// SIMATIC S7-200 project (STEP 7-Micro/WIN), CPU 224XP CN REL 02.01

SYMBOL_TABLE 用户定义1
键值输出1            I0.0
键值输出2            I0.1
键值输出3            I0.2
键值输出4            I0.3
传感器输出A           I0.4
传感器输出B           I0.5
传感器输出C           I0.6
传感器输出D           I0.7
手自动              I1.0
启停               I1.1
位置显示A            Q0.0
位置显示B            Q0.1
位置显示C            Q0.2
正传左行             Q0.3
反转右行             Q0.4
快速               Q0.5
慢速               Q0.6
报警               Q0.7
END_SYMBOL_TABLE

ORGANIZATION_BLOCK 主程序:OB1
TITLE=小车运动1A
// V0.0进入初始复位子程序控制位
// V0.1进入手动子程序控制位
// V0.2进入自动子程序控制位
// VW10初始复位控制用
// VW20手动控制用
// VW30自动控制用
BEGIN
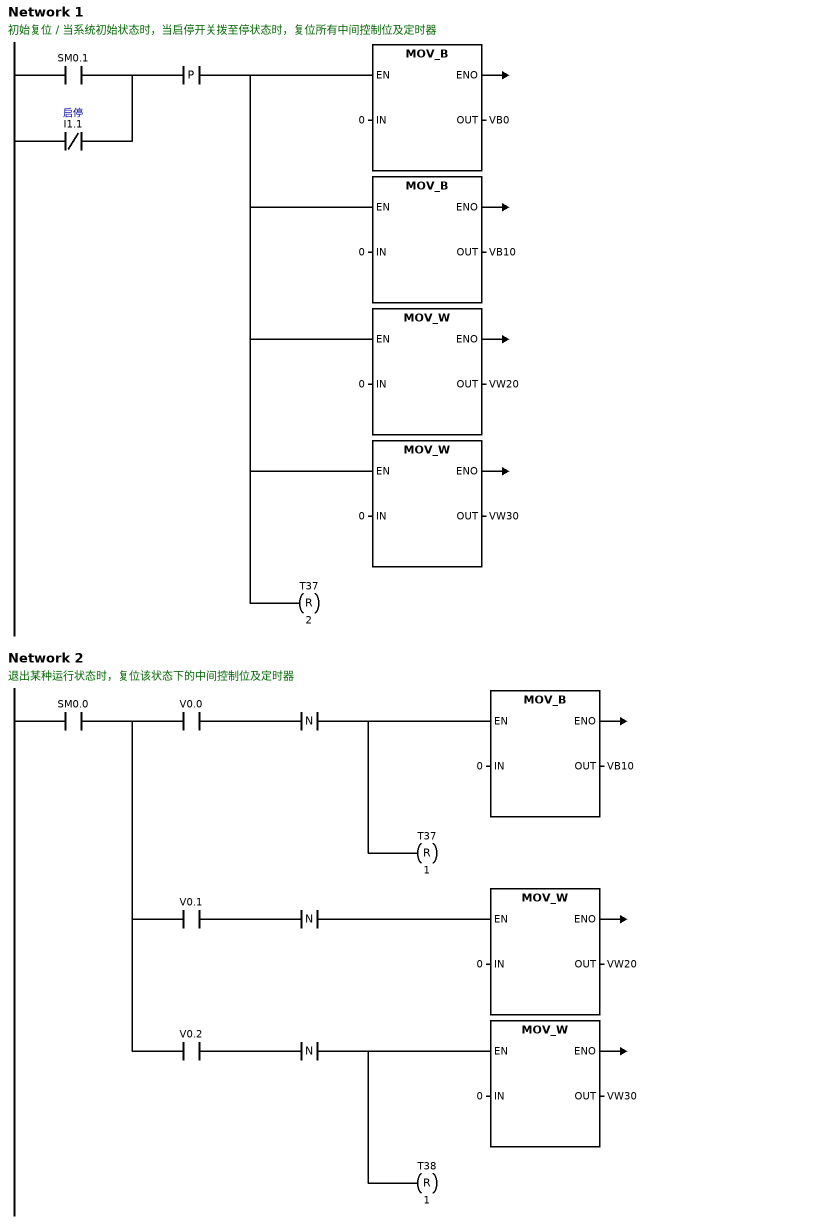
Network 1
// 初始复位
// 当系统初始状态时，当启停开关拨至停状态时，复位所有中间控制位及定时器
LD     SM0.1
ON     启停:I1.1
EU
MOVB   0, VB0
MOVB   0, VB10
MOVW   0, VW20
MOVW   0, VW30
R      T37, 2
Network 2
// 退出某种运行状态时，复位该状态下的中间控制位及定时器
LD     SM0.0
LPS
A      V0.0
ED
MOVB   0, VB10
R      T37, 1
LRD
A      V0.1
ED
MOVW   0, VW20
LPP
A      V0.2
ED
MOVW   0, VW30
R      T38, 1
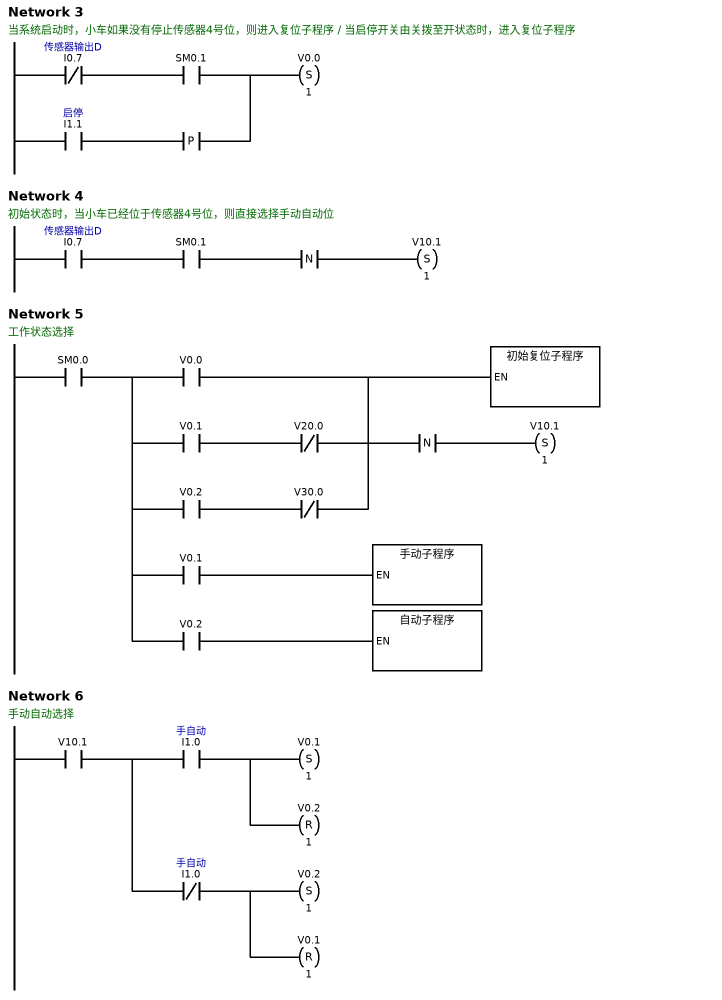
Network 3
// 当系统启动时，小车如果没有停止传感器4号位，则进入复位子程序
// 当启停开关由关拨至开状态时，进入复位子程序
LDN    传感器输出D:I0.7
A      SM0.1
LD     启停:I1.1
EU
OLD
S      V0.0, 1
Network 4
// 初始状态时，当小车已经位于传感器4号位，则直接选择手动自动位
LD     传感器输出D:I0.7
A      SM0.1
ED
S      V10.1, 1
Network 5
// 工作状态选择
LD     SM0.0
LPS
LD     V0.0
LD     V0.1
AN     V20.0
OLD
LD     V0.2
AN     V30.0
OLD
ALD
CALL   初始复位子程序:SBR0
ED
S      V10.1, 1
LPP
LPS
A      V0.1
CALL   手动子程序:SBR1
LPP
A      V0.2
CALL   自动子程序:SBR2
Network 6
// 手动自动选择
LD     V10.1
LPS
A      手自动:I1.0
S      V0.1, 1
R      V0.2, 1
LPP
AN     手自动:I1.0
S      V0.2, 1
R      V0.1, 1
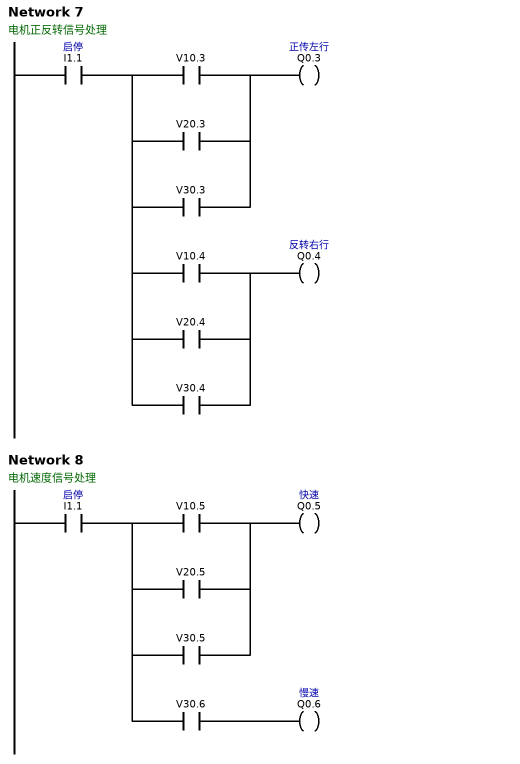
Network 7
// 电机正反转信号处理
LD     启停:I1.1
LPS
LD     V10.3
O      V20.3
O      V30.3
ALD
=      正传左行:Q0.3
LPP
LD     V10.4
O      V20.4
O      V30.4
ALD
=      反转右行:Q0.4
Network 8
// 电机速度信号处理
LD     启停:I1.1
LPS
LD     V10.5
O      V20.5
O      V30.5
ALD
=      快速:Q0.5
LPP
A      V30.6
=      慢速:Q0.6
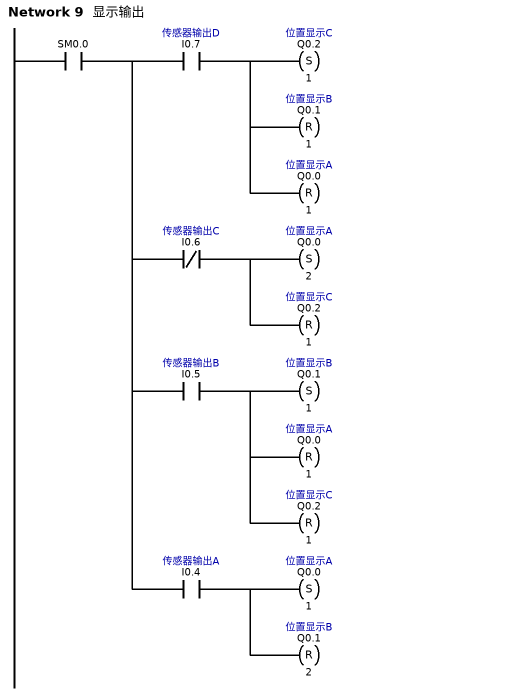
Network 9 // 显示输出
LD     SM0.0
LPS
A      传感器输出D:I0.7
S      位置显示C:Q0.2, 1
R      位置显示B:Q0.1, 1
R      位置显示A:Q0.0, 1
LRD
AN     传感器输出C:I0.6
S      位置显示A:Q0.0, 2
R      位置显示C:Q0.2, 1
LRD
A      传感器输出B:I0.5
S      位置显示B:Q0.1, 1
R      位置显示A:Q0.0, 1
R      位置显示C:Q0.2, 1
LPP
A      传感器输出A:I0.4
S      位置显示A:Q0.0, 1
R      位置显示B:Q0.1, 2
END_ORGANIZATION_BLOCK

SUBROUTINE_BLOCK 初始复位子程序:SBR0
TITLE=子程序注释
BEGIN
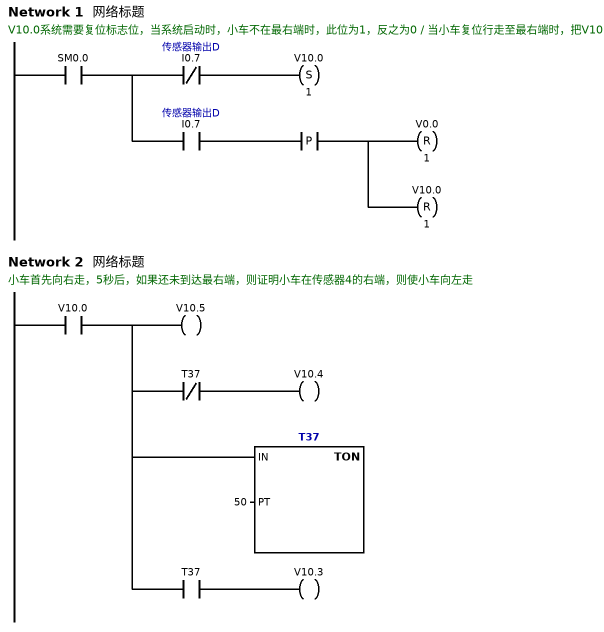
Network 1 // 网络标题
// V10.0系统需要复位标志位，当系统启动时，小车不在最右端时，此位为1，反之为0
// 当小车复位行走至最右端时，把V10.0复位，把调用子程序有效位V0.0复位。
LD     SM0.0
LPS
AN     传感器输出D:I0.7
S      V10.0, 1
LPP
A      传感器输出D:I0.7
EU
R      V0.0, 1
R      V10.0, 1
Network 2 // 网络标题
// 小车首先向右走，5秒后，如果还未到达最右端，则证明小车在传感器4的右端，则使小车向左走
LD     V10.0
LPS
=      V10.5
AN     T37
=      V10.4
LRD
TON    T37, 50
LPP
A      T37
=      V10.3
END_SUBROUTINE_BLOCK

SUBROUTINE_BLOCK 手动子程序:SBR1
TITLE=子程序注释
BEGIN
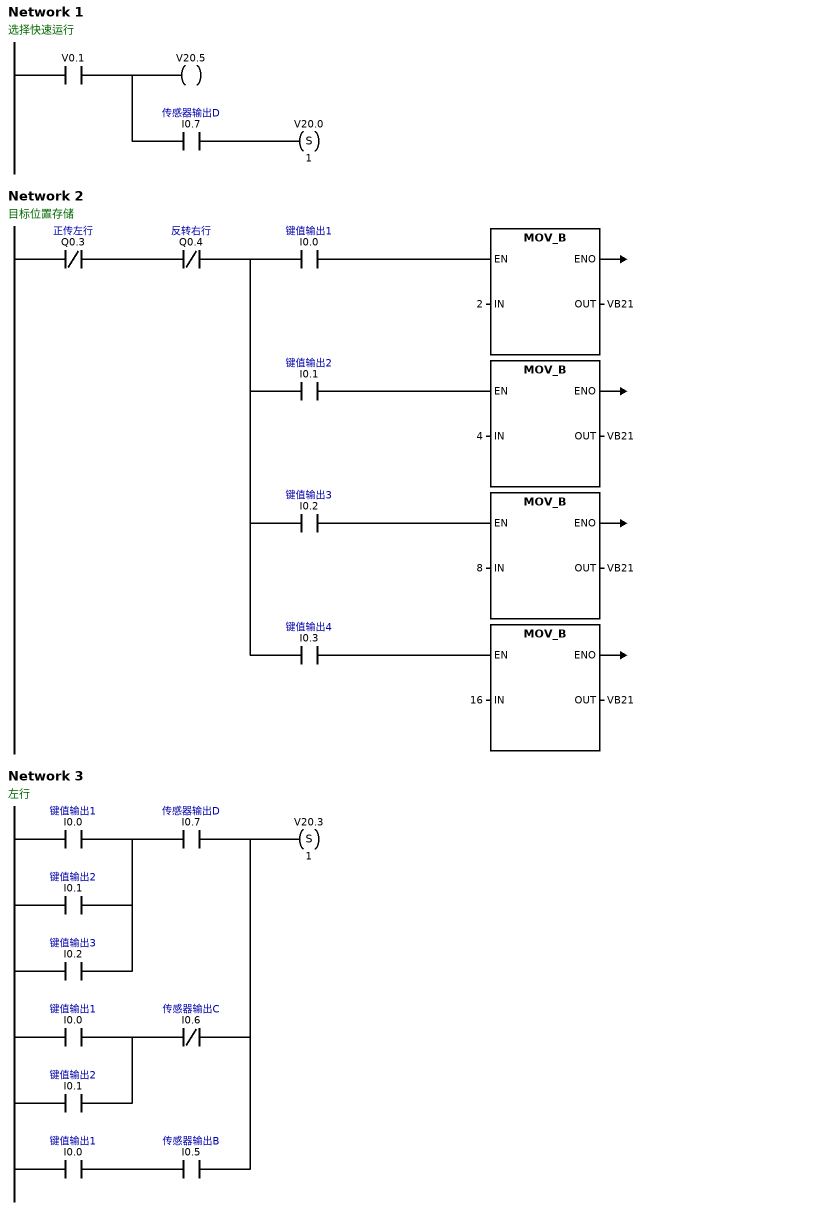
Network 1
// 选择快速运行
LD     V0.1
=      V20.5
A      传感器输出D:I0.7
S      V20.0, 1
Network 2
// 目标位置存储
LDN    正传左行:Q0.3
AN     反转右行:Q0.4
LPS
A      键值输出1:I0.0
MOVB   2, VB21
LRD
A      键值输出2:I0.1
MOVB   4, VB21
LRD
A      键值输出3:I0.2
MOVB   8, VB21
LPP
A      键值输出4:I0.3
MOVB   16, VB21
Network 3
// 左行
LD     键值输出1:I0.0
O      键值输出2:I0.1
O      键值输出3:I0.2
A      传感器输出D:I0.7
LD     键值输出1:I0.0
O      键值输出2:I0.1
AN     传感器输出C:I0.6
OLD
LD     键值输出1:I0.0
A      传感器输出B:I0.5
OLD
S      V20.3, 1
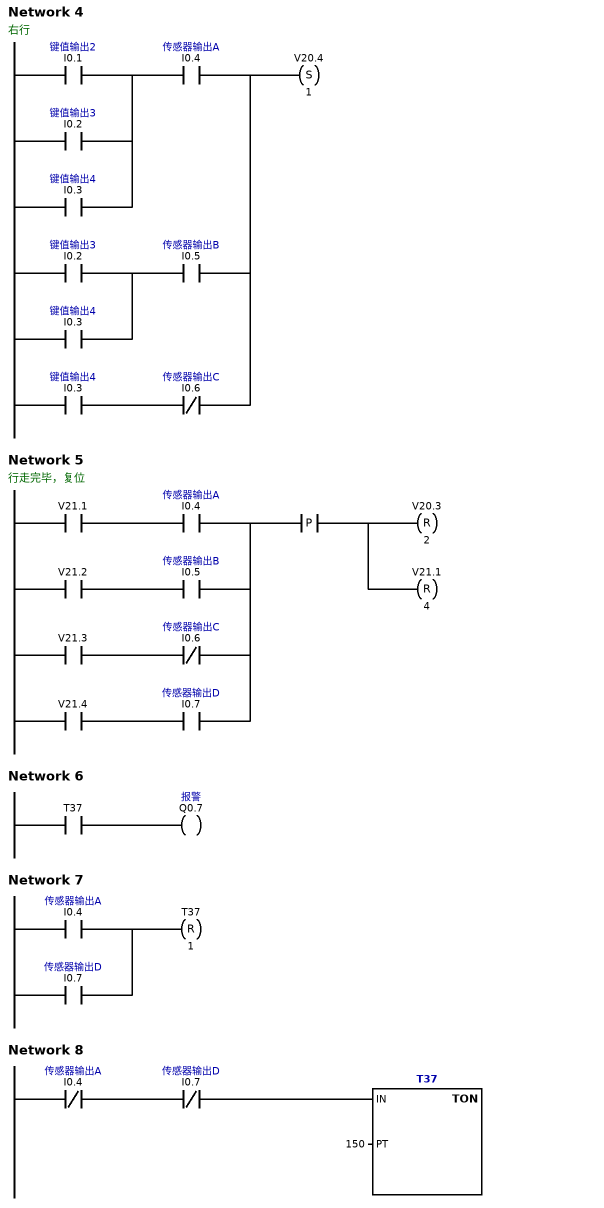
Network 4
// 右行
LD     键值输出2:I0.1
O      键值输出3:I0.2
O      键值输出4:I0.3
A      传感器输出A:I0.4
LD     键值输出3:I0.2
O      键值输出4:I0.3
A      传感器输出B:I0.5
OLD
LD     键值输出4:I0.3
AN     传感器输出C:I0.6
OLD
S      V20.4, 1
Network 5
// 行走完毕，复位
LD     V21.1
A      传感器输出A:I0.4
LD     V21.2
A      传感器输出B:I0.5
OLD
LD     V21.3
AN     传感器输出C:I0.6
OLD
LD     V21.4
A      传感器输出D:I0.7
OLD
EU
R      V20.3, 2
R      V21.1, 4
Network 6
LD     T37
=      报警:Q0.7
Network 7
LD     传感器输出A:I0.4
O      传感器输出D:I0.7
R      T37, 1
Network 8
LDN    传感器输出A:I0.4
AN     传感器输出D:I0.7
TON    T37, 150
END_SUBROUTINE_BLOCK

SUBROUTINE_BLOCK 自动子程序:SBR2
TITLE=子程序注释
BEGIN
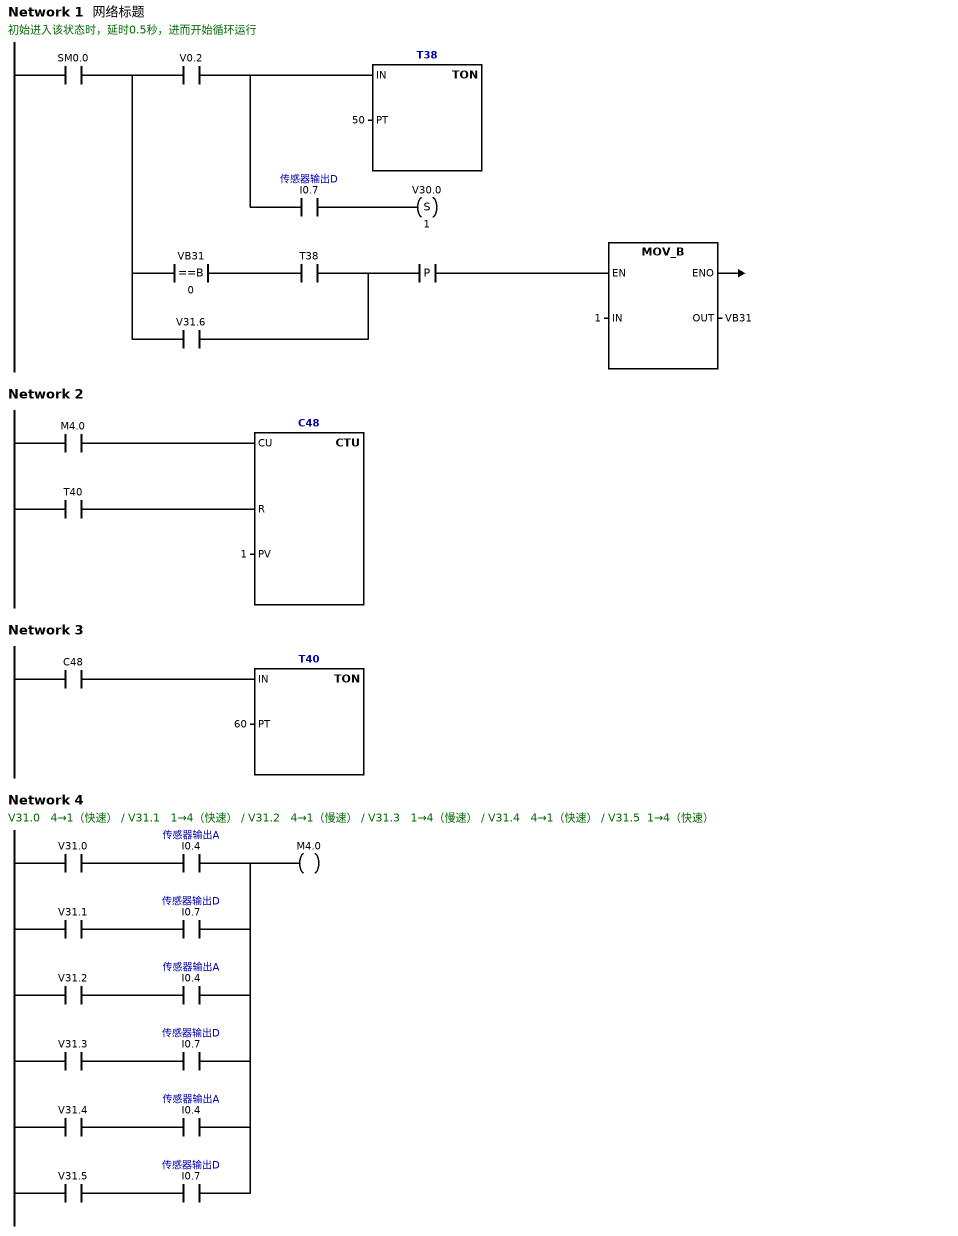
Network 1 // 网络标题
// 初始进入该状态时，延时0.5秒，进而开始循环运行
LD     SM0.0
LPS
A      V0.2
TON    T38, 50
A      传感器输出D:I0.7
S      V30.0, 1
LPP
LDB=   VB31, 0
A      T38
O      V31.6
ALD
EU
MOVB   1, VB31
Network 2
LD     M4.0
LD     T40
CTU    C48, 1
Network 3
LD     C48
TON    T40, 60
Network 4
// V31.0   4→1（快速）
// V31.1   1→4（快速）
// V31.2   4→1（慢速）
// V31.3   1→4（慢速）
// V31.4   4→1（快速）
// V31.5  1→4（快速）
LD     V31.0
A      传感器输出A:I0.4
LD     V31.1
A      传感器输出D:I0.7
OLD
LD     V31.2
A      传感器输出A:I0.4
OLD
LD     V31.3
A      传感器输出D:I0.7
OLD
LD     V31.4
A      传感器输出A:I0.4
OLD
LD     V31.5
A      传感器输出D:I0.7
OLD
=      M4.0
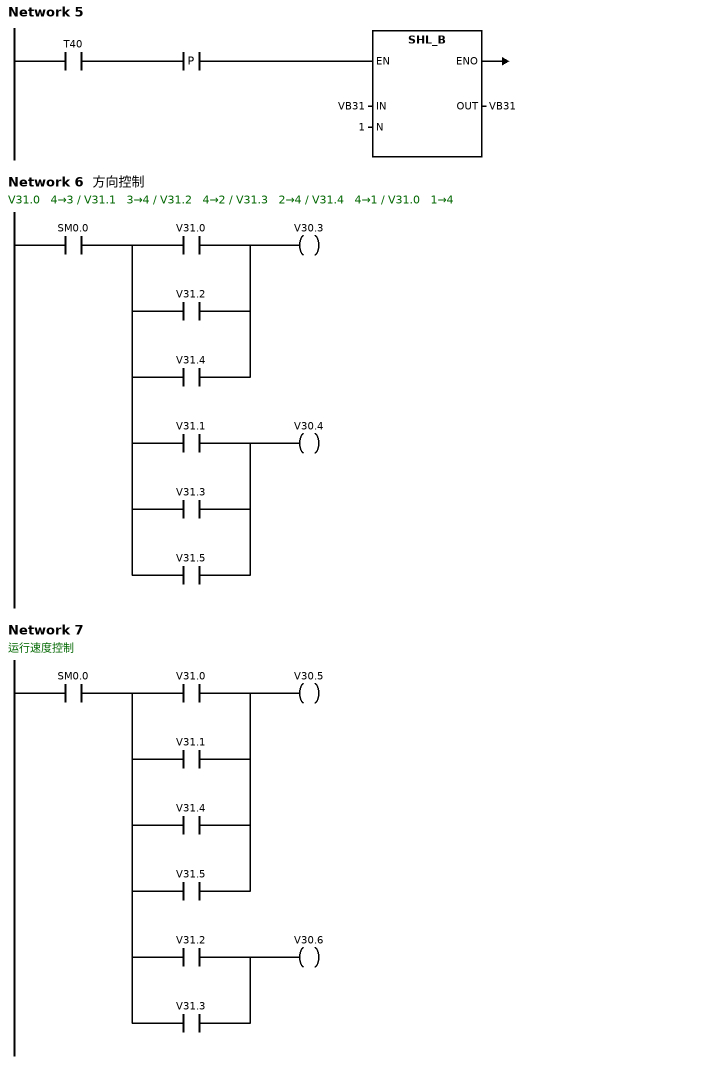
Network 5
LD     T40
EU
SLB    VB31, 1
Network 6 // 方向控制
// V31.0   4→3
// V31.1   3→4
// V31.2   4→2
// V31.3   2→4
// V31.4   4→1
// V31.0   1→4
LD     SM0.0
LPS
LD     V31.0
O      V31.2
O      V31.4
ALD
=      V30.3
LPP
LD     V31.1
O      V31.3
O      V31.5
ALD
=      V30.4
Network 7
// 运行速度控制
LD     SM0.0
LPS
LD     V31.0
O      V31.1
O      V31.4
O      V31.5
ALD
=      V30.5
LPP
LD     V31.2
O      V31.3
ALD
=      V30.6
END_SUBROUTINE_BLOCK
